FUNCTION_BLOCK ABSTRACT FB_Logger IMPLEMENTS I_Logger
VAR_INPUT
END_VAR
VAR_OUTPUT
END_VAR
VAR
	stParameter:		ST_Logger;
END_VAR

METHOD M_Critical
VAR_INPUT
	Message	: STRING(255);
END_VAR
END_METHOD

METHOD M_Debug
VAR_INPUT
	Message	: STRING(255);
END_VAR
END_METHOD

METHOD M_Error
VAR_INPUT
	Message:		STRING(255);
END_VAR
END_METHOD

METHOD M_Info
VAR_INPUT
	Message	: STRING(255);
END_VAR
END_METHOD

METHOD M_Log
VAR_INPUT
	LogLevel:		E_LogLevel;
	Message:		STRING(255);
END_VAR
END_METHOD

METHOD M_Warning
VAR_INPUT
	Message	: STRING(255);
END_VAR
END_METHOD

PROPERTY PUBLIC P_Parameter : reference to ST_Logger
GET
END_GET
END_PROPERTY

END_FUNCTION_BLOCK

(* stored: Version 1.1.0.1
   POU FB_Logger: Id {75e85e1a-2f6e-03ab-0c87-a271e0cb3059}, SpecialFunc None
   Method M_Critical: Id {2c8a5c1c-03ce-0010-0a47-0212c31c090a}
   Method M_Debug: Id {e3912c08-cf4d-007c-00c3-1ee82a0d186f}
   Method M_Error: Id {03bff8e4-5538-0253-230e-ccdcab79aad4}
   Method M_Info: Id {2ddc58e6-49ca-01d6-1dfd-87a9538cab59}
   Method M_Log: Id {4452c859-b6bf-01af-3dbe-b917edbc909d}
   Method M_Warning: Id {0990c154-baa1-08fc-1e9d-e8bdc2ce38cc}
   Property P_Parameter: Id {c3786a2f-91e3-0ec1-3f7a-a85190472496}
   Get Get: Id {5db43e1f-632d-0054-2947-dbccd362cd17} *)
